FUNCTION_BLOCK FB_EtherCATTopologyDiagnosis
VAR_INPUT
END_VAR
VAR_OUTPUT
END_VAR
VAR
END_VAR

END_FUNCTION_BLOCK

(* stored: Version 1.1.0.1, ProductVersion 3.1.4026.18
   POU FB_EtherCATTopologyDiagnosis: Id {6fe1c4c8-cec6-4d64-a8c8-dffaa5ef8150}, SpecialFunc None *)
